ABB RobotStudio station: RS_proyecto_G1E1.rsstn

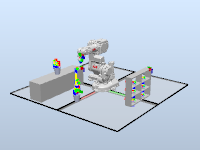
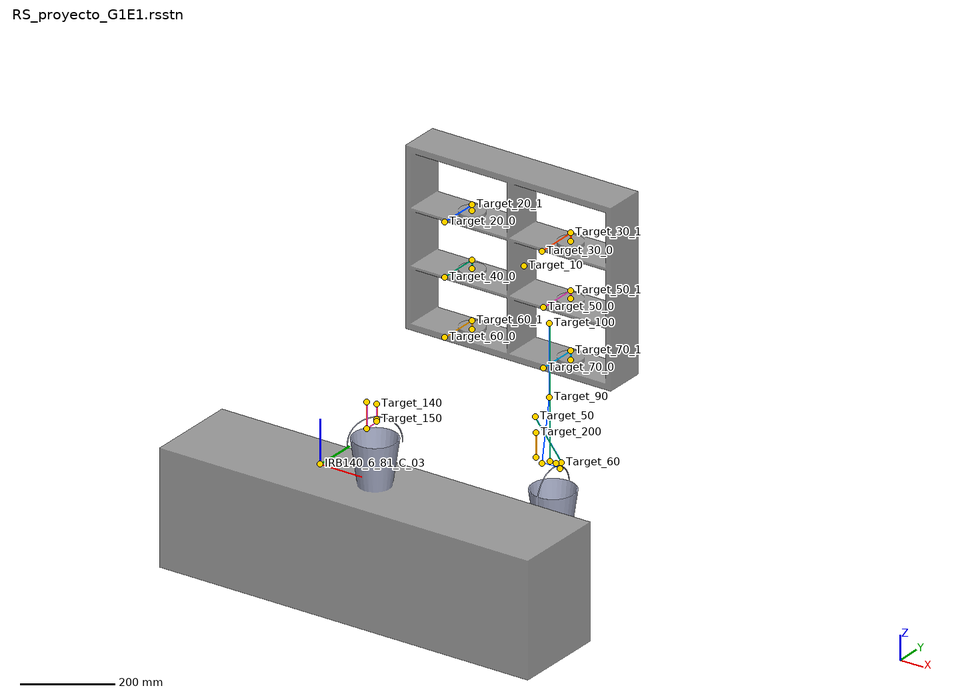
[picture v1: parts stored in the station drawn from their meshes, with robot base, taught points and paths (robot models come from the ABB library and are not in the file)]
Station proyecto (saved by RobotStudio 22.1.9826.0)
Controller Controller1
  mechanical unit ROB_1: IRB140_6_81_C_03, 6 joints, base frame (0, 0, 0) mm
Layout (positions relative to the parent item):
  - IRB140_6_81_C_03 [mechanism, from Robots\IRB140_6_81_C_G_03.rslib] at (0, 0, 0) mm; joint values [0, 0, 0, 0, 0.5236, 0] (rad or m)
  - VentosaTool [mechanism, from Libraries\VentosaTool.rslib] at (506.29, 0, 679.5) mm, rotated rx 180 ry 60 rz 180 deg
  - BANDA [part] at (480, -600, 140) mm, rotated rx 0 ry -90 rz 0 deg, size 280 x 230 x 950 mm
  - Gabinete [part] at (300, 740.64, 0) mm, rotated rx -90 ry 0 rz -90 deg, size 100 x 430 x 530 mm
  - Monedas_2 [part] at (162, 690.64, 286) mm, rotated rx 90 ry 0 rz 0 deg, size 60 x 10 x 59.7 mm
  - Monedas_3 [part] at (-92, 690.64, 150) mm, rotated rx 90 ry 0 rz 0 deg, size 60 x 10 x 59.7 mm
  - Monedas_4 [part] at (162, 690.64, 150) mm, rotated rx 90 ry 0 rz 0 deg, size 60 x 10 x 59.7 mm
  - Monedas_5 [part] at (-92, 690.64, 14) mm, rotated rx 90 ry 0 rz 0 deg, size 60 x 10 x 59.7 mm
  - Monedas_6 [part] at (162, 690.64, 14) mm, rotated rx 90 ry 0 rz 0 deg, size 60 x 10 x 59.7 mm
  - Monedas_1 [part] at (-92, 690.64, 286) mm, rotated rx 90 ry 0 rz 0 deg, size 60 x 10 x 59.7 mm
  - Valde [part] at (600, 0, 0) mm, rotated rx 90 ry 0 rz 0 deg, size 106 x 161 x 120.6 mm
  - GanchoToolPlus [mechanism, from Libraries\GanchoToolPlus.rslib] at (506.29, 0, 679.5) mm, rotated rx 180 ry 60 rz 180 deg
  - Valde_2 [part] at (480, -485, 280) mm, rotated rx 90 ry 0 rz 135 deg, size 106 x 161 x 120.6 mm
Attachment: VentosaTool is attached to IRB140_6_81_C_03 / Link6
Attachment: GanchoToolPlus is attached to IRB140_6_81_C_03 / Link6
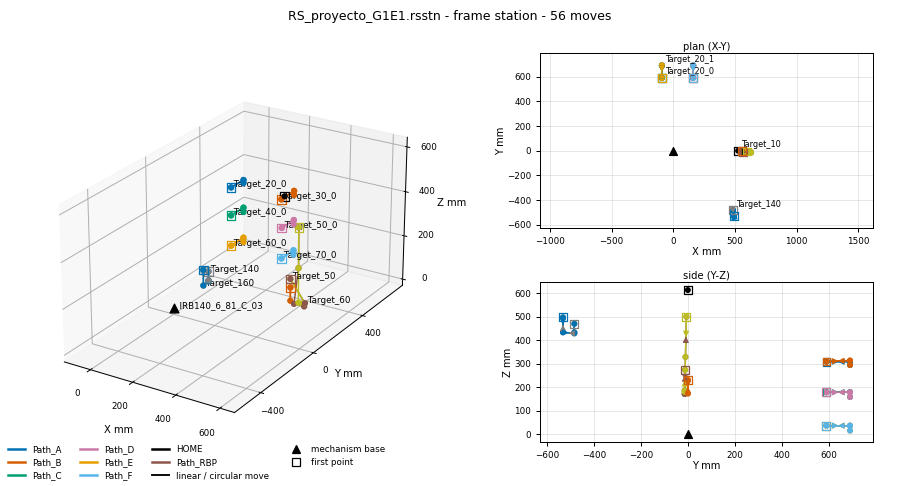
[picture p0: tool path of RS_proyecto_G1E1.rsstn in frame station, 56 of 56 moves have a stored position in this frame; points joined in program order, loops and branches not executed]
Targets, tools, work objects and paths stored in the station, written as RAPID:
! task T_ROB1
MODULE CalibData
  PERS tooldata VentosaToolTCP:=[TRUE,[[47.334,0,50],[0.707106781,0,0.707106781,0]],[2,[5.462,-4.903,-3.606],[1,0,0,0],0,0,0]];
  TASK PERS wobjdata GabineteWobj:=[FALSE,TRUE,"",[[-36.5,0,-2],[1,0,0,0]],[[-193.694,740.638,430],[0,1,0,0]]];
  TASK PERS wobjdata BaldeWobj:=[FALSE,TRUE,"",[[0,0,30],[1,0,0,0]],[[548.980124364,-0.000124471,110.279],[1,0,0,0.000000001]]];
  PERS tooldata GanchoToolPlus:=[TRUE,[[-0.129,37.5,33],[0.5,-0.5,0.5,0.5]],[1,[5.242,15,47.094],[1,0,0,0],0,0,0]];
  TASK PERS wobjdata BandaWobj:=[FALSE,TRUE,"",[[5,-370,280],[0,1,0,0]],[[0,0,0],[1,0,0,0]]];
ENDMODULE

! task T_ROB1
MODULE Module1
  CONST robtarget Target_10:=[[525.925921435,0,613.507553537],[0.258819045,0,-0.965925826,0],[0,0,0,0],[9E+09,9E+09,9E+09,9E+09,9E+09,9E+09]];
  CONST robtarget Target_40_2:=[[138.194,50,270],[0.707106781,0,0,0.707106781],[1,0,-1,1],[9E+09,9E+09,9E+09,9E+09,9E+09,9E+09]];
  CONST robtarget Target_50_2:=[[392.194,50,270],[0.707106781,0,0,0.707106781],[0,-1,0,1],[9E+09,9E+09,9E+09,9E+09,9E+09,9E+09]];
  CONST robtarget Target_60_2:=[[138.194,50,413],[0.707106781,0,0,0.707106781],[1,0,-1,1],[9E+09,9E+09,9E+09,9E+09,9E+09,9E+09]];
  CONST robtarget Target_70_2:=[[392.194,50,413],[0.707106781,0,0,0.707106781],[0,-1,0,1],[9E+09,9E+09,9E+09,9E+09,9E+09,9E+09]];
  CONST robtarget Target_40_1:=[[138.193999586,50.000010178,249.329325634],[0.707106779,-0.000000008,0.000000037,0.707106783],[1,0,-1,1],[9E+09,9E+09,9E+09,9E+09,9E+09,9E+09]];
  CONST robtarget Target_40_0:=[[138.194021584,150.352701404,249.329292581],[0.707106793,0.000000006,0.000000022,0.70710677],[1,0,-1,1],[9E+09,9E+09,9E+09,9E+09,9E+09,9E+09]];
  CONST robtarget Target_50_1:=[[392.193956988,50.000000319,249.860330541],[0.70710676,-0.000000006,0.000000021,0.707106802],[0,-1,0,1],[9E+09,9E+09,9E+09,9E+09,9E+09,9E+09]];
  CONST robtarget Target_50_0:=[[392.193987544,150.452485445,249.860309256],[0.707106776,-0.000000001,0.000000048,0.707106787],[0,-1,0,1],[9E+09,9E+09,9E+09,9E+09,9E+09,9E+09]];
  CONST robtarget Target_70_1:=[[392.194037432,50.000013786,391.930189862],[0.707106799,0.000000016,-0.000000035,0.707106764],[0,-1,0,1],[9E+09,9E+09,9E+09,9E+09,9E+09,9E+09]];
  CONST robtarget Target_70_0:=[[392.194001399,150.543672268,391.930177073],[0.707106781,-0.000000034,-0.000000042,0.707106781],[0,-1,0,1],[9E+09,9E+09,9E+09,9E+09,9E+09,9E+09]];
  CONST robtarget Target_60_1:=[[138.193996276,49.999994893,391.734498057],[0.707106782,-0.000000048,-0.000000042,0.70710678],[1,0,-1,1],[9E+09,9E+09,9E+09,9E+09,9E+09,9E+09]];
  CONST robtarget Target_60_0:=[[138.193995129,150.580831923,391.734551119],[0.707106782,-0.000000033,0.000000006,0.70710678],[1,0,-1,1],[9E+09,9E+09,9E+09,9E+09,9E+09,9E+09]];
  CONST robtarget Target_20_0:=[[138.194017242,150.352702998,119.277210229],[0.707106777,-0.000000038,0.000000034,0.707106785],[1,0,-1,1],[9E+09,9E+09,9E+09,9E+09,9E+09,9E+09]];
  CONST robtarget Target_20_2:=[[138.194,50,134],[0.707106781,0,0,0.707106781],[1,0,-1,1],[9E+09,9E+09,9E+09,9E+09,9E+09,9E+09]];
  CONST robtarget Target_20_1:=[[138.194067358,50.000000634,119.720304143],[0.707106782,-0.000000015,0.000000001,0.70710678],[1,0,-1,1],[9E+09,9E+09,9E+09,9E+09,9E+09,9E+09]];
  CONST robtarget Target_30_0:=[[388.906866606,150.352702732,118.620023306],[0.707106792,0.00000006,0.000000045,0.707106771],[0,-1,0,1],[9E+09,9E+09,9E+09,9E+09,9E+09,9E+09]];
  CONST robtarget Target_30_2:=[[392.194,50,134],[0.707106781,0,0,0.707106781],[0,-1,0,1],[9E+09,9E+09,9E+09,9E+09,9E+09,9E+09]];
  CONST robtarget Target_30_1:=[[392.194040299,50.00000744,114.731091406],[0.707106756,0.000000008,-0.000000024,0.707106806],[0,-1,0,1],[9E+09,9E+09,9E+09,9E+09,9E+09,9E+09]];
  CONST robtarget Target_3:=[[51.019875636,0.000124369,20],[0,0.000000001,1,0],[0,0,0,0],[9E+09,9E+09,9E+09,9E+09,9E+09,9E+09]];
  CONST robtarget Target_1:=[[-57.601324247,0.000124586,25.900391186],[0.000000021,0.707106782,0.70710678,-0.000000021],[0,0,0,1],[9E+09,9E+09,9E+09,9E+09,9E+09,9E+09]];
  CONST robtarget Target_2:=[[51.148337293,0.000124369,25.900385765],[-0.000000045,0.000000001,1,0],[0,0,0,1],[9E+09,9E+09,9E+09,9E+09,9E+09,9E+09]];
  CONST robtarget Target_50:=[[13.302672904,-11.431256176,133.30348639],[0.01014685,0.000116761,0.999875397,-0.012092072],[-1,-1,-2,1],[9E+09,9E+09,9E+09,9E+09,9E+09,9E+09]];
  CONST robtarget Target_60:=[[82.19086006,-13.579085665,45.862304116],[0.010146855,0.000116761,0.999875397,-0.012092063],[-1,-1,-2,1],[9E+09,9E+09,9E+09,9E+09,9E+09,9E+09]];
  CONST robtarget Target_70:=[[68.860686652,-13.696344759,40.749981845],[0.010146861,0.000116762,0.999875397,-0.012092085],[-1,-1,-2,1],[9E+09,9E+09,9E+09,9E+09,9E+09,9E+09]];
  CONST robtarget Target_80:=[[52.254489531,-13.696543478,40.412904783],[0.010146879,0.000116762,0.999875397,-0.012092065],[-1,-1,-2,1],[9E+09,9E+09,9E+09,9E+09,9E+09,9E+09]];
  CONST robtarget Target_90:=[[49.251846553,-10.117436033,188.337190497],[0.010146904,0.000116761,0.999875397,-0.012092046],[-1,-1,-2,1],[9E+09,9E+09,9E+09,9E+09,9E+09,9E+09]];
  CONST robtarget Target_100:=[[45.773262616,-5.97116956,359.702605623],[0.010146919,0.000116761,0.999875397,-0.012092056],[-1,-1,-2,1],[9E+09,9E+09,9E+09,9E+09,9E+09,9E+09]];
  CONST robtarget Target_130:=[[475,115,-110.279],[0.382683433,0,0,-0.923879532],[0,0,0,0],[9E+09,9E+09,9E+09,9E+09,9E+09,9E+09]];
  CONST robtarget Target_140:=[[478.854792248,113.143397052,-189.978969725],[0.409457701,-0.005060563,-0.013507452,-0.912215068],[-1,0,-2,1],[9E+09,9E+09,9E+09,9E+09,9E+09,9E+09]];
  CONST robtarget Target_150:=[[478.85479121,113.143395442,-153.35140145],[0.409457704,-0.005060601,-0.013507452,-0.912215067],[-1,0,-2,1],[9E+09,9E+09,9E+09,9E+09,9E+09,9E+09]];
  CONST robtarget Target_160:=[[487.269593662,161.6317163,-153.351393014],[0.409457704,-0.005060634,-0.013507406,-0.912215067],[-1,0,-2,1],[9E+09,9E+09,9E+09,9E+09,9E+09,9E+09]];
  CONST robtarget Target_170:=[[487.269594744,161.631715665,-217.285689258],[0.409457703,-0.00506064,-0.013507396,-0.912215068],[-1,0,-2,1],[9E+09,9E+09,9E+09,9E+09,9E+09,9E+09]];
  CONST robtarget Target_180:=[[478.854791357,113.143395609,-148.949893987],[0.409457703,-0.00506064,-0.01350747,-0.912215067],[-1,0,-2,1],[9E+09,9E+09,9E+09,9E+09,9E+09,9E+09]];
  CONST robtarget Target_210:=[[6.878996642,0.591031162,31.883291445],[0.003025406,0.71249878,-0.013165639,0.7015433],[0,-2,-1,1],[9E+09,9E+09,9E+09,9E+09,9E+09,9E+09]];
  CONST robtarget Target_200:=[[6.878987614,0.591034871,89.637373996],[0.003025441,0.712498803,-0.013165757,0.701543274],[0,-2,0,1],[9E+09,9E+09,9E+09,9E+09,9E+09,9E+09]];
  CONST robtarget Target_220:=[[78.860695651,-13.69634493,30.749995921],[0.01014684,0.000116762,0.999875397,-0.012092069],[-1,-1,-2,1],[9E+09,9E+09,9E+09,9E+09,9E+09,9E+09]];
  CONST robtarget Target_230:=[[32.254479792,-13.696545985,30.412884885],[0.010146873,0.000116761,0.999875397,-0.012092092],[-1,-1,-2,1],[9E+09,9E+09,9E+09,9E+09,9E+09,9E+09]];
  PROC Path_A()
    MoveJ Target_20_0,v300,z100,VentosaToolTCP\WObj:=GabineteWobj;
    MoveL Target_20_1,v100,z100,VentosaToolTCP\WObj:=GabineteWobj;
    MoveL Target_20_2,v100,z100,VentosaToolTCP\WObj:=GabineteWobj;
    MoveL Target_20_1,v100,z100,VentosaToolTCP\WObj:=GabineteWobj;
    MoveL Target_20_0,v100,z100,VentosaToolTCP\WObj:=GabineteWobj;
  ENDPROC
  PROC Path_B()
    MoveJ Target_30_0,v300,z100,VentosaToolTCP\WObj:=GabineteWobj;
    MoveL Target_30_1,v100,z100,VentosaToolTCP\WObj:=GabineteWobj;
    MoveL Target_30_2,v100,z100,VentosaToolTCP\WObj:=GabineteWobj;
    MoveL Target_30_1,v100,z100,VentosaToolTCP\WObj:=GabineteWobj;
    MoveL Target_30_0,v100,z100,VentosaToolTCP\WObj:=GabineteWobj;
  ENDPROC
  PROC Path_C()
    MoveJ Target_40_0,v300,z100,VentosaToolTCP\WObj:=GabineteWobj;
    MoveL Target_40_1,v100,z100,VentosaToolTCP\WObj:=GabineteWobj;
    MoveL Target_40_2,v100,z100,VentosaToolTCP\WObj:=GabineteWobj;
    MoveL Target_40_1,v100,z100,VentosaToolTCP\WObj:=GabineteWobj;
    MoveL Target_40_0,v100,z100,VentosaToolTCP\WObj:=GabineteWobj;
  ENDPROC
  PROC Path_D()
    MoveJ Target_50_0,v300,z100,VentosaToolTCP\WObj:=GabineteWobj;
    MoveL Target_50_1,v100,z100,VentosaToolTCP\WObj:=GabineteWobj;
    MoveL Target_50_2,v100,z100,VentosaToolTCP\WObj:=GabineteWobj;
    MoveL Target_50_1,v100,z100,VentosaToolTCP\WObj:=GabineteWobj;
    MoveL Target_50_0,v100,z100,VentosaToolTCP\WObj:=GabineteWobj;
  ENDPROC
  PROC Path_E()
    MoveJ Target_60_0,v300,z100,VentosaToolTCP\WObj:=GabineteWobj;
    MoveL Target_60_1,v100,z100,VentosaToolTCP\WObj:=GabineteWobj;
    MoveL Target_60_2,v100,z100,VentosaToolTCP\WObj:=GabineteWobj;
    MoveL Target_60_1,v100,z100,VentosaToolTCP\WObj:=GabineteWobj;
    MoveL Target_60_0,v100,z100,VentosaToolTCP\WObj:=GabineteWobj;
  ENDPROC
  PROC Path_F()
    MoveJ Target_70_0,v300,z100,VentosaToolTCP\WObj:=GabineteWobj;
    MoveL Target_70_1,v100,z100,VentosaToolTCP\WObj:=GabineteWobj;
    MoveL Target_70_2,v100,z100,VentosaToolTCP\WObj:=GabineteWobj;
    MoveL Target_70_1,v100,z100,VentosaToolTCP\WObj:=GabineteWobj;
    MoveL Target_70_0,v100,z100,VentosaToolTCP\WObj:=GabineteWobj;
  ENDPROC
  PROC HOME()
    MoveJ Target_10,v300,z100,VentosaToolTCP\WObj:=wobj0;
  ENDPROC
  PROC Path_RBP()
    MoveJ Target_50,v300,z100,GanchoToolPlus\WObj:=BaldeWobj;
    MoveL Target_60,v100,z100,GanchoToolPlus\WObj:=BaldeWobj;
    MoveL Target_220,v100,z100,GanchoToolPlus\WObj:=BaldeWobj;
    MoveL Target_230,v100,z100,GanchoToolPlus\WObj:=BaldeWobj;
    MoveL Target_90,v100,z100,GanchoToolPlus\WObj:=BaldeWobj;
    MoveL Target_100,v100,z100,GanchoToolPlus\WObj:=BaldeWobj;
  ENDPROC
  PROC Path_DBB()
    MoveJ Target_140,v200,z100,GanchoToolPlus\WObj:=BandaWobj;
    MoveL Target_150,v100,z100,GanchoToolPlus\WObj:=BandaWobj;
    MoveL Target_180,v100,z100,GanchoToolPlus\WObj:=BandaWobj;
    MoveL Target_160,v100,z100,GanchoToolPlus\WObj:=BandaWobj;
    MoveL Target_170,v100,z100,GanchoToolPlus\WObj:=BandaWobj;
  ENDPROC
  PROC Path_DBP()
    MoveJ Target_100,v100,z100,GanchoToolPlus\WObj:=BaldeWobj;
    MoveL Target_90,v100,z100,GanchoToolPlus\WObj:=BaldeWobj;
    MoveL Target_80,v100,z100,GanchoToolPlus\WObj:=BaldeWobj;
    MoveL Target_70,v100,z100,GanchoToolPlus\WObj:=BaldeWobj;
    MoveL Target_60,v100,z100,GanchoToolPlus\WObj:=BaldeWobj;
    MoveL Target_50,v100,z100,GanchoToolPlus\WObj:=BaldeWobj;
  ENDPROC
  PROC Path_RBB()
    MoveJ Target_170,v300,z100,GanchoToolPlus\WObj:=BandaWobj;
    MoveL Target_160,v100,z100,GanchoToolPlus\WObj:=BandaWobj;
    MoveL Target_180,v100,z100,GanchoToolPlus\WObj:=BandaWobj;
    MoveL Target_150,v100,z100,GanchoToolPlus\WObj:=BandaWobj;
    MoveL Target_140,v100,z100,GanchoToolPlus\WObj:=BandaWobj;
  ENDPROC
  PROC Path_Deposito()
    MoveJ Target_200,v300,z100,VentosaToolTCP\WObj:=BaldeWobj;
    MoveL Target_210,v100,z100,VentosaToolTCP\WObj:=BaldeWobj;
    MoveL Target_200,v200,z100,VentosaToolTCP\WObj:=BaldeWobj;
  ENDPROC
ENDMODULE

